TYPE Socket :
STRUCT
	localAdr : T_AmsNetId;
	localPort : T_AmsPort;
	
	remoteAdr : T_AmsNetId;
	remotePort : T_AmsPort;
END_STRUCT
END_TYPE

(* stored: Version 1.1.0.1, ProductVersion 3.1.4024.11
   DUT Socket: Id {c910e2ed-3567-4ea4-b927-59a7d3ae026b} *)
